// TIA Portal V20 export
// export: Created 2025-12-01T14:57:06.9577599Z, ExportSetting None, DisplayName Totally Integrated Automation Portal, DisplayVersion V20 Update 3, DisplayName TIA Portal Openness, DisplayVersion V20 Update 3, DisplayName TIA Portal Version Control Interface, DisplayVersion V20 Update 3, DisplayName STEP 7 Professional, DisplayVersion V20 Update 3, DisplayName STEP 7 Safety, DisplayVersion V20 Update 2, DisplayName WinCC Basic/Comfort/Advanced, DisplayVersion V20 Update 3, DisplayName WinCC Professional, DisplayVersion V20 Update 3, DisplayName WinCC Unified, DisplayVersion V20 Update 3
FUNCTION "FC986_CRTL_VAR_LENZE_Remo" : Void   // FC986, LAD
{ S7_Optimized_Access := 'FALSE' }
AUTHOR : LENZE
NAME : 20130301
VERSION : 3.0
// stored: AutoNumber false, SetENOAutomatically false
   VAR_INPUT
      Byte_Inicial : Int;
      Esclavo_NO_PRESENTE : Bool;
      Sacar_Horquilla : Bool;
      Recoger_Horquilla : Bool;
      Subir_Horquilla : Bool;
      Bajar_Horquilla : Bool;
      Rearme_T : Bool;
      Selector_Mvto : Bool;
      Fallo_Externo : Bool;
      Fr_Consigna : Word;
   END_VAR
   VAR_IN_OUT
      VarLenze : "UDT_VarLenze";
   END_VAR
   VAR_TEMP
      STW : Struct   // Codigo de Estado
         IN_Libre_8 : Bool;   // Bit coded display of the active device state
         IN_Libre_9 : Bool;   // Bit coded display of the active device state
         IN_Libre_10 : Bool;   // Bit coded display of the active device state
         IN_Libre_11 : Bool;   // Bit coded display of the active device state
         IN_Libre_12 : Bool;   // 1 = A warning exists.
         IN_Libre_13 : Bool;   // 1 = Controller is in the "Trouble" device state
         IN_Libre_14 : Bool;   // Direction of rotation: 0 = Clockwise (Cw), 1 = Counter-clockwise (Ccw)
         IN_Libre_15 : Bool;   // 1 = Drive controller is ready for operation
         IN_DriveFail : Bool;
         IN_DriveReady : Bool;   // 1 = Inverter control inhibited (pulse inhibit is active)
         IN_InhActive : Bool;
         IN_QSP_Active : Bool;
         IN_SentidoGiro : Bool;
         IN_Zero_Speed : Bool;
         IN_IMax_Active : Bool;   // 1 = Current speed is 0
         IN_SelecParam : Bool;   // 1 = Controller inhibited (controller inhibit is active)
      END_STRUCT;
      CTW : Struct   // Codigo de Control
         Out_Libre_8 : Bool;   // 1 = Activate stop function. Stop drive via stopping ramp.
         Out_Libre_9 : Bool;
         Out_Libre_10 : Bool;
         Out_Libre_11 : Bool;   // 1 = Activate DC-injection braking
         Out_Libre_12 : Bool;
         Out_Libre_13 : Bool;
         Out_Libre_14 : Bool;   // 1 = Set error (trip set)
         Out_Libre_15 : Bool;   // 0 = To the right (Cw), 1 = To the left (Ccw)
         Out_Inhvir_Var : Bool;   // 1 = Change to the "SwitchedON" device state
         Out_Rearme_Var : Bool;   // 1 = Inhibit inverter control (IMP - pulse inhibit)
         Out_Set_Quick_Stop : Bool;   // 1 = Activate quick stop (QSP).
         Out_Sentido_Giro : Bool;   // 1 = Enable controller (RFR)
         Out_CambioParam : Bool;
         Out_Libre_5 : Bool;
         Out_Libre_6 : Bool;
         Out_Libre_7 : Bool;   // 1 = Reset fault (trip reset)
      END_STRUCT;
      MRV : Word;   // Consigna
      Temp_Consigna : DInt;
      P_Variador : DWord;
      P_STW : DWord;
      P_CTW : DWord;
   END_VAR
BEGIN

REGION Network 1: SI NO ESTA EL NODO, SALTAMOS AL FINAL PARA NO JODER CICLO SCAN
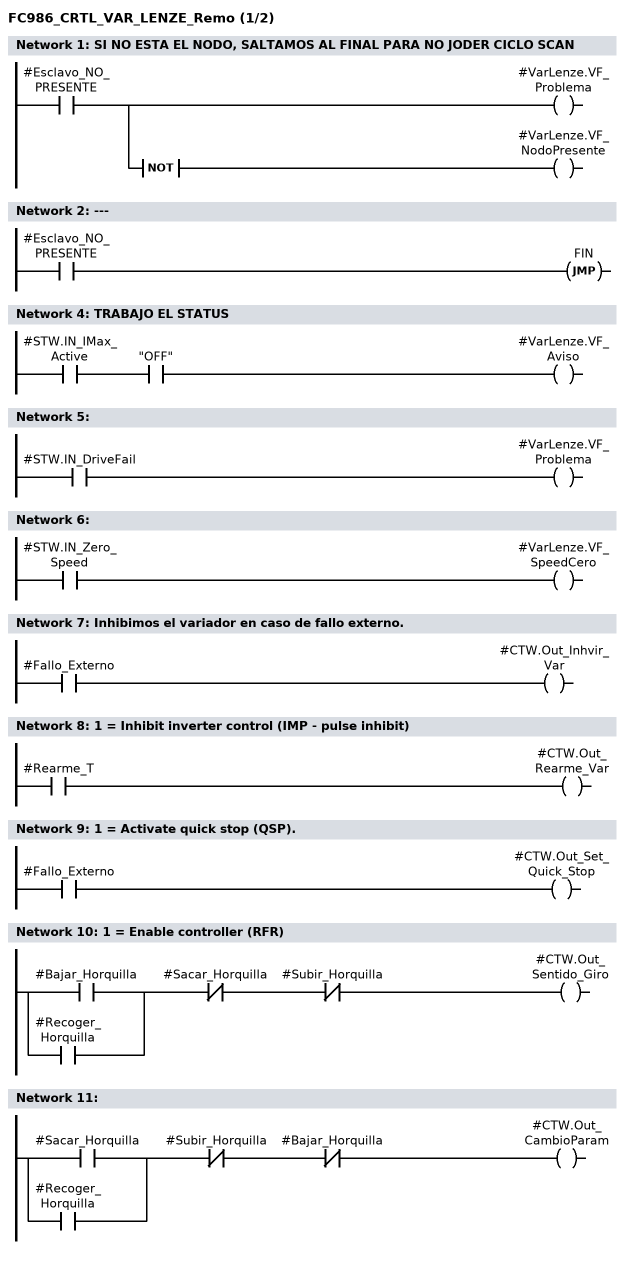
   RUNG wire#powerrail
      Contact( #Esclavo_NO_PRESENTE )
      wire#w1
      Coil( #VarLenze.VF_Problema )
   END_RUNG
   RUNG wire#w1
      Not()
      Coil( #VarLenze.VF_NodoPresente )
   END_RUNG
   // the same network as SCL:
   #VarLenze.VF_Problema := #Esclavo_NO_PRESENTE;
   #VarLenze.VF_NodoPresente := NOT #Esclavo_NO_PRESENTE;
END_REGION

REGION Network 2: ---
   RUNG wire#powerrail
      Contact( #Esclavo_NO_PRESENTE )
      JumpCoil( FIN )
   END_RUNG
   // the same network as SCL:
   IF #Esclavo_NO_PRESENTE THEN GOTO FIN; END_IF;
END_REGION

NETWORK
TITLE = LECTURA WORD ESTADO VARIADOR Y PASO A BITs SALIDA
//==============================================
//=====                                    =====
//===== Created by:  Jokin Altuna          =====
//=====                 22/06/2012         =====
//==============================================


      L     P##STW;  // Punteros
      T     #P_STW;
      L     P##CTW;
      T     #P_CTW;

//==============================================
      L     #Byte_Inicial;  //Obtener Direccion Inicio PEW
      SLD   3;  //Dar formato de Integer a Puntero
      LAR1;  //Guardar en el Registro 1

//==============================================

      L     IW [AR1, P#2.0];  //Cargar primer Word de Status
      T     LW [#P_STW];  //Guardamos en temporal para manejar bits.

//==============================================

REGION Network 4: TRABAJO EL STATUS
   RUNG wire#powerrail
      Contact( #STW.IN_IMax_Active )
      Contact( "OFF" )
      Coil( #VarLenze.VF_Aviso )
   END_RUNG
   // the same network as SCL:
   #VarLenze.VF_Aviso := #STW.IN_IMax_Active AND "OFF";
END_REGION

REGION Network 5
   RUNG wire#powerrail
      Contact( #STW.IN_DriveFail )
      Coil( #VarLenze.VF_Problema )
   END_RUNG
   // the same network as SCL:
   #VarLenze.VF_Problema := #STW.IN_DriveFail;
END_REGION

REGION Network 6
   RUNG wire#powerrail
      Contact( #STW.IN_Zero_Speed )
      Coil( #VarLenze.VF_SpeedCero )
   END_RUNG
   // the same network as SCL:
   #VarLenze.VF_SpeedCero := #STW.IN_Zero_Speed;
END_REGION

REGION Network 7: Inhibimos el variador en caso de fallo externo.
   RUNG wire#powerrail
      Contact( #Fallo_Externo )
      Coil( #CTW.Out_Inhvir_Var )
   END_RUNG
   // the same network as SCL:
   #CTW.Out_Inhvir_Var := #Fallo_Externo;
END_REGION

REGION Network 8: 1 = Inhibit inverter control (IMP - pulse inhibit)
   RUNG wire#powerrail
      Contact( #Rearme_T )
      Coil( #CTW.Out_Rearme_Var )
   END_RUNG
   // the same network as SCL:
   #CTW.Out_Rearme_Var := #Rearme_T;
END_REGION

REGION Network 9: 1 = Activate quick stop (QSP).
   RUNG wire#powerrail
      Contact( #Fallo_Externo )
      Coil( #CTW.Out_Set_Quick_Stop )
   END_RUNG
   // the same network as SCL:
   #CTW.Out_Set_Quick_Stop := #Fallo_Externo;
END_REGION

REGION Network 10: 1 = Enable controller (RFR)
   RUNG wire#powerrail
      Contact( #Bajar_Horquilla )
      wire#w1
      I_Contact( #Sacar_Horquilla )
      I_Contact( #Subir_Horquilla )
      Coil( #CTW.Out_Sentido_Giro )
   END_RUNG
   RUNG wire#powerrail
      Contact( #Recoger_Horquilla )
   END_RUNG wire#w1
   // the same network as SCL:
   #CTW.Out_Sentido_Giro := (#Bajar_Horquilla OR #Recoger_Horquilla) AND NOT #Sacar_Horquilla AND NOT #Subir_Horquilla;
END_REGION

REGION Network 11
   RUNG wire#powerrail
      Contact( #Sacar_Horquilla )
      wire#w1
      I_Contact( #Subir_Horquilla )
      I_Contact( #Bajar_Horquilla )
      Coil( #CTW.Out_CambioParam )
   END_RUNG
   RUNG wire#powerrail
      Contact( #Recoger_Horquilla )
   END_RUNG wire#w1
   // the same network as SCL:
   #CTW.Out_CambioParam := (#Sacar_Horquilla OR #Recoger_Horquilla) AND NOT #Subir_Horquilla AND NOT #Bajar_Horquilla;
END_REGION

REGION Network 12
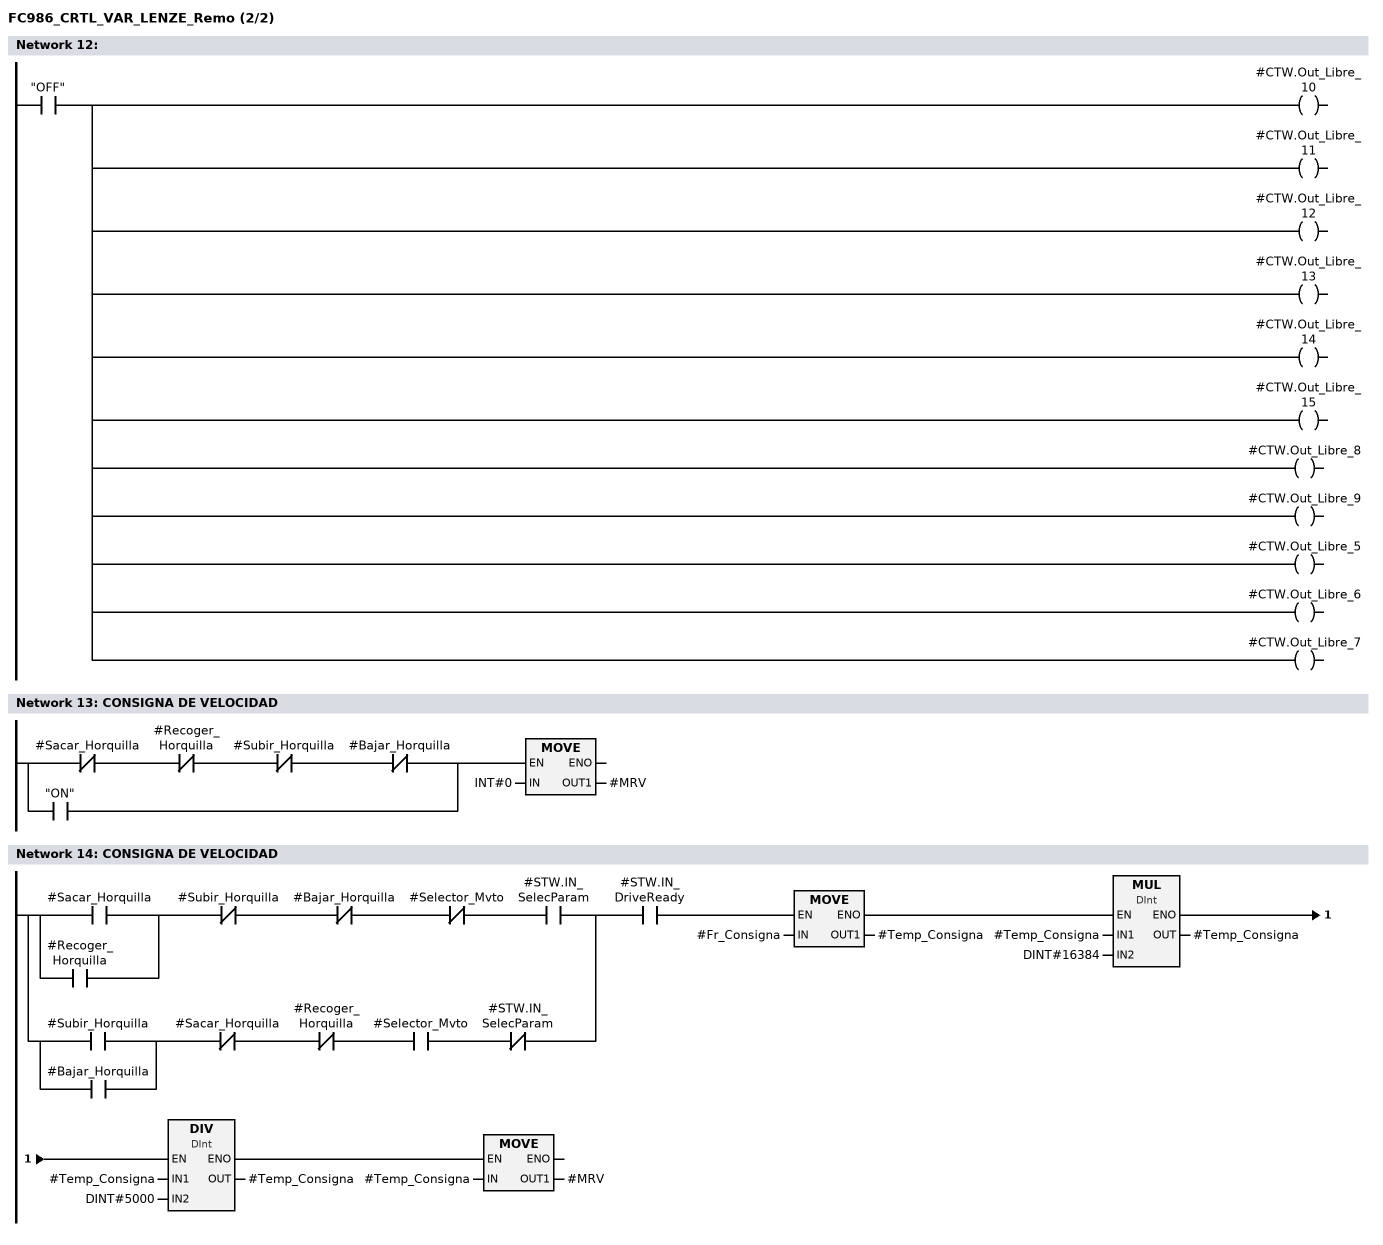
   RUNG wire#powerrail
      Contact( "OFF" )
      wire#w1
      Coil( #CTW.Out_Libre_10 )
   END_RUNG
   RUNG wire#w1
      Coil( #CTW.Out_Libre_11 )
   END_RUNG
   RUNG wire#w1
      Coil( #CTW.Out_Libre_12 )
   END_RUNG
   RUNG wire#w1
      Coil( #CTW.Out_Libre_13 )
   END_RUNG
   RUNG wire#w1
      Coil( #CTW.Out_Libre_14 )
   END_RUNG
   RUNG wire#w1
      Coil( #CTW.Out_Libre_15 )
   END_RUNG
   RUNG wire#w1
      Coil( #CTW.Out_Libre_8 )
   END_RUNG
   RUNG wire#w1
      Coil( #CTW.Out_Libre_9 )
   END_RUNG
   RUNG wire#w1
      Coil( #CTW.Out_Libre_5 )
   END_RUNG
   RUNG wire#w1
      Coil( #CTW.Out_Libre_6 )
   END_RUNG
   RUNG wire#w1
      Coil( #CTW.Out_Libre_7 )
   END_RUNG
   // the same network as SCL:
   #CTW.Out_Libre_10 := "OFF";
   #CTW.Out_Libre_11 := "OFF";
   #CTW.Out_Libre_12 := "OFF";
   #CTW.Out_Libre_13 := "OFF";
   #CTW.Out_Libre_14 := "OFF";
   #CTW.Out_Libre_15 := "OFF";
   #CTW.Out_Libre_8 := "OFF";
   #CTW.Out_Libre_9 := "OFF";
   #CTW.Out_Libre_5 := "OFF";
   #CTW.Out_Libre_6 := "OFF";
   #CTW.Out_Libre_7 := "OFF";
END_REGION

REGION Network 13: CONSIGNA DE VELOCIDAD
   RUNG wire#powerrail
      I_Contact( #Sacar_Horquilla )
      I_Contact( #Recoger_Horquilla )
      I_Contact( #Subir_Horquilla )
      I_Contact( #Bajar_Horquilla )
      wire#w1
      { S7_GenerateENO := "TRUE" } Move(in := INT#0, out1 => #MRV)
   END_RUNG
   RUNG wire#powerrail
      Contact( "ON" )
   END_RUNG wire#w1
   // the same network as SCL:
   IF (NOT #Sacar_Horquilla AND NOT #Recoger_Horquilla AND NOT #Subir_Horquilla AND NOT #Bajar_Horquilla) OR "ON" THEN
       #MRV := INT#0;
   END_IF;
END_REGION

REGION Network 14: CONSIGNA DE VELOCIDAD
   RUNG wire#powerrail
      Contact( #Sacar_Horquilla )
      wire#w1
      I_Contact( #Subir_Horquilla )
      I_Contact( #Bajar_Horquilla )
      I_Contact( #Selector_Mvto )
      Contact( #STW.IN_SelecParam )
      wire#w2
      Contact( #STW.IN_DriveReady )
      { S7_GenerateENO := "TRUE" } Move(in := #Fr_Consigna, out1 => #Temp_Consigna)
      { S7_Templates := "SrcType := DInt"; S7_GenerateENO := "TRUE" } Mul(in1 := #Temp_Consigna, in2 := DINT#16384, out => #Temp_Consigna)
      { S7_Templates := "SrcType := DInt"; S7_GenerateENO := "TRUE" } Div(in1 := #Temp_Consigna, in2 := DINT#5000, out => #Temp_Consigna)
      { S7_GenerateENO := "TRUE" } Move(in := #Temp_Consigna, out1 => #MRV)
   END_RUNG
   RUNG wire#powerrail
      Contact( #Recoger_Horquilla )
   END_RUNG wire#w1
   RUNG wire#powerrail
      Contact( #Subir_Horquilla )
      wire#w3
      I_Contact( #Sacar_Horquilla )
      I_Contact( #Recoger_Horquilla )
      Contact( #Selector_Mvto )
      I_Contact( #STW.IN_SelecParam )
   END_RUNG wire#w2
   RUNG wire#powerrail
      Contact( #Bajar_Horquilla )
   END_RUNG wire#w3
   // the same network as SCL:
   // ENO of a box is taken as its EN; it also drops when the box reports an error
   IF (((#Sacar_Horquilla OR #Recoger_Horquilla) AND NOT #Subir_Horquilla AND NOT #Bajar_Horquilla AND NOT #Selector_Mvto AND #STW.IN_SelecParam) OR ((#Subir_Horquilla OR #Bajar_Horquilla) AND NOT #Sacar_Horquilla AND NOT #Recoger_Horquilla AND #Selector_Mvto AND NOT #STW.IN_SelecParam)) AND #STW.IN_DriveReady THEN
       #Temp_Consigna := #Fr_Consigna;
       #Temp_Consigna := #Temp_Consigna * DINT#16384;
       #Temp_Consigna := #Temp_Consigna / DINT#5000;
       #MRV := #Temp_Consigna;
   END_IF;
END_REGION

NETWORK
TITLE = ESCRITURA WORD CONTROL VARIADOR
//======================================
      L     #Byte_Inicial;  //Obtener Direccion Inicio PAW
      SLD   3;  //Dar formato de Integer a Puntero
      LAR1;  //Guardar en el Registro 1
//=======================================
      L     LW [#P_CTW];  //Carga valores de salida
      T     QW [AR1, P#2.0];  //Transfiere a salida Profibus

      L     #MRV;
      T     QW [AR1, P#4.0];



NETWORK
TITLE = 
FIN:  NOP   0;


END_FUNCTION
